{attribute 'qualified_only'}
VAR_GLOBAL CONSTANT
	cServiceCount : UINT := SIZEOF(ST_Chamber1_ServiceCtrl) / SIZEOF(ST_ServiceCtrl);
END_VAR

(* stored: Version 1.1.0.1, ProductVersion 3.1.4026.18
   GVL GVL_Chamber1_Config: Id {e17c4bd1-c3da-471b-9592-c1512b9dedb8} *)
